(* PLC project tanks_management, Dassault Systèmes ControlBuild 2024x *)
(* stored: creationDateTime 2023-10-03T11:13:41-01:00 *)

FUNCTION_BLOCK bottling_line.tanks_management
  VAR_INPUT
    productionRequest : BOOL := false;
    closingRequest : BOOL := false;
    masterInStandBy : BOOL := false;
  END_VAR
  VAR_INPUT
    highLevel1 : BOOL := false;
    highLevel2 : BOOL := false;
    highLevel3 : BOOL := false;
  END_VAR
  VAR_INPUT
    lowLevel1 : BOOL := false;
    lowLevel2 : BOOL := false;
    lowLevel3 : BOOL := false;
  END_VAR
  VAR_OUTPUT
    pump1 : BOOL := false;
    pump2 : BOOL := false;
    valve1 : BOOL := false;
    valve2 : BOOL := false;
    valve3 : BOOL := false;
    valve4 : BOOL := false;
    lowSpeedAgitator : BOOL := false;
    highSpeedAgitator : BOOL := false;
  END_VAR
  VAR_OUTPUT
    closingEnd : BOOL := false;
  END_VAR

INITIAL_STEP 10:
  COMPUTE_FUNCTION_BLOCKS(S);
END_STEP
TRANSITION FROM 10 TO 11
  := productionRequest OR closingRequest;
END_TRANSITION
INITIAL_STEP 20:
END_STEP
TRANSITION FROM 20 TO 21
  := productionRequest AND lowLevel1;
END_TRANSITION
INITIAL_STEP 30:
END_STEP
TRANSITION FROM 30 TO 31
  := productionRequest AND lowLevel2;
END_TRANSITION
STEP 11:
  11_INLINE1(N);
END_STEP
ACTION 11_INLINE1:
  lowSpeedAgitator;
END_ACTION
TRANSITION FROM 11 TO 12
  := lowLevel3 AND NOT lowLevel1 AND NOT lowLevel2 AND productionRequest OR closingRequest;
END_TRANSITION
STEP 21:
  21_INLINE2(N);
END_STEP
ACTION 21_INLINE2:
  valve1;
END_ACTION
TRANSITION FROM 21 TO 20
  := highLevel1 OR NOT productionRequest;
END_TRANSITION
STEP 12:
  12_INLINE3(N);
END_STEP
ACTION 12_INLINE3:
  highSpeedAgitator;
  pump1;
  pump2;
  valve3;
  valve4;
END_ACTION
TRANSITION FROM 12 TO 13
  := highLevel3 OR lowLevel1 OR lowLevel2 OR NOT (productionRequest AND closingRequest );
END_TRANSITION
STEP 13:
  13_INLINE4(N);
END_STEP
ACTION 13_INLINE4:
  closingEnd;
END_ACTION
TRANSITION FROM 13 TO 10
  := masterInStandBy;
END_TRANSITION
STEP 31:
  31_INLINE5(N);
END_STEP
ACTION 31_INLINE5:
  valve2;
END_ACTION
TRANSITION FROM 31 TO 30
  := highLevel2 OR NOT productionRequest;
END_TRANSITION
ACTION COMPUTE_FUNCTION_BLOCKS:  (* blocks drawn on the SFC sheet *)
  G1:
  G2:
  G3:
END_ACTION
END_FUNCTION_BLOCK
